INTERFACE I_XTS_Group  EXTENDS I_CH_Object

METHOD AddAxisListToGroup : HRESULT
VAR_INPUT
	ipMovers : I_CH_List;
END_VAR
END_METHOD

METHOD AddingAxisToGroup : HRESULT
END_METHOD

PROPERTY AllAxesStanding : Bool
GET
END_GET
END_PROPERTY

METHOD ChangeGapMode : HRESULT
VAR_INPUT
	bFast : BOOL;
END_VAR
END_METHOD

METHOD Disable : HRESULT
VAR_INPUT
END_VAR
END_METHOD

METHOD Enable : HRESULT
VAR_INPUT
END_VAR
END_METHOD

{attribute 'monitoring':='call'}
PROPERTY GroupEnabled : BOOL
GET
END_GET
END_PROPERTY

{attribute 'monitoring':='call'}
PROPERTY HR : HRESULT
GET
END_GET
END_PROPERTY

METHOD Initialize : HRESULT
VAR_INPUT
END_VAR
END_METHOD

METHOD RemoveAxisFromGroup : HRESULT
VAR_INPUT
	ipMover : I_XTS_Mover;
END_VAR
END_METHOD

METHOD Reset : HRESULT
VAR_INPUT
END_VAR
END_METHOD

METHOD UngroupAllAxes : HRESULT
VAR_INPUT
END_VAR
END_METHOD

METHOD Update : HRESULT
VAR_INPUT
END_VAR
END_METHOD

{attribute 'monitoring':='call'}
PROPERTY UtilityCAGroup : I_Mc2CaGroup
GET
END_GET
END_PROPERTY

END_INTERFACE

(* stored: Version 1.1.0.1, ProductVersion 3.1.4024.12
   Itf I_XTS_Group: Id {3aa79aea-eed3-48e5-9919-147a82f1dcae}
   Method AddAxisListToGroup: Id {14ba38af-55d1-438e-87b3-bcb9deeb2c08}
   Method AddingAxisToGroup: Id {15bb7821-6d23-406e-8575-4d183a93525a}
   Property AllAxesStanding: Id {18b8de0f-763c-4967-b374-93d6f61fbccc}
   Get Get: Id {93882710-e532-48df-a654-6f38816b3433}
   Method ChangeGapMode: Id {53b260d0-0e84-422c-bdf9-45d5721e6a88}
   Method Disable: Id {49a59ea7-a3d9-4b46-895b-593b3e02df7c}
   Method Enable: Id {1b778060-30cb-4774-8cdb-b397b8102027}
   Property GroupEnabled: Id {fe8dbb55-e36a-4328-baaa-b3c17dbcf20e}
   Get Get: Id {9af12953-3591-4bd2-a3b7-484b60d9650f}
   Property HR: Id {531b6a0c-8750-4388-b1bc-f79833a91add}
   Get Get: Id {20a7df7f-4ea8-45e0-bc93-01d51e482e82}
   Method Initialize: Id {97c43364-5a87-4076-9341-9fd384ac3f88}
   Method RemoveAxisFromGroup: Id {ae50f6db-1093-4586-8191-72a2fb88fe19}
   Method Reset: Id {0a246b89-9fb9-4319-9113-6eb69b6d818e}
   Method UngroupAllAxes: Id {95ad16a3-687a-4192-a41d-ae3a71ea2284}
   Method Update: Id {3d7c5dc0-7d33-45d1-920d-34225572deeb}
   Property UtilityCAGroup: Id {a9fc9959-e685-4084-8d82-b3e62e08ab6f}
   Get Get: Id {88e70f16-e941-4f3c-b9b2-3386c05d27cd} *)
